PROGRAM MAIN
VAR
	axis1: AXIS_REF;
	axis2: AXIS_REF;
	axis3: AXIS_REF;
	
	delay: TON;
	powerAxis1: MC_Power;
	moveAxis1: MC_MoveVelocity;
	resetAxis1: MC_Reset;
	
	enableControl: BOOL	:=0;
	enablePos: BOOL		:=0;
	enableNeg: BOOL		:=0;
	override: LREAL		:=0;
	active: BOOL		:=0;
	direction: INT		:=0;
	execute: BOOL		:=0;

	state: INT			:=0;
	nextState:INT		:=0;

END_VAR


axis1.ReadStatus();
//axis2.ReadStatus();
//axis3.ReadStatus();

enableControl:=1;
enablePos:=1;
enableNeg:=1;
override:=100;
execute:=0;

powerAxis1(Axis:=axis1,Enable:=enableControl,Enable_Positive:=enablePos,Enable_Negative:=enableNeg,Override:=override);

IF powerAxis1.Active THEN
	delay(IN:=powerAxis1.Active,PT:=T#500MS);
END_IF
IF delay.Q THEN
	execute:=1;
	moveAxis1(Axis:=axis1,Velocity:=250,Direction:=MC_Positive_Direction,Execute:=execute,BufferMode:=MC_Buffered);
END_IF

END_PROGRAM

(* stored: Version 1.1.0.1, ProductVersion 3.1.4022.3
   POU MAIN: Id {e82fe949-bc40-4bc0-b1a4-f8ef83395fe3}, SpecialFunc None *)
